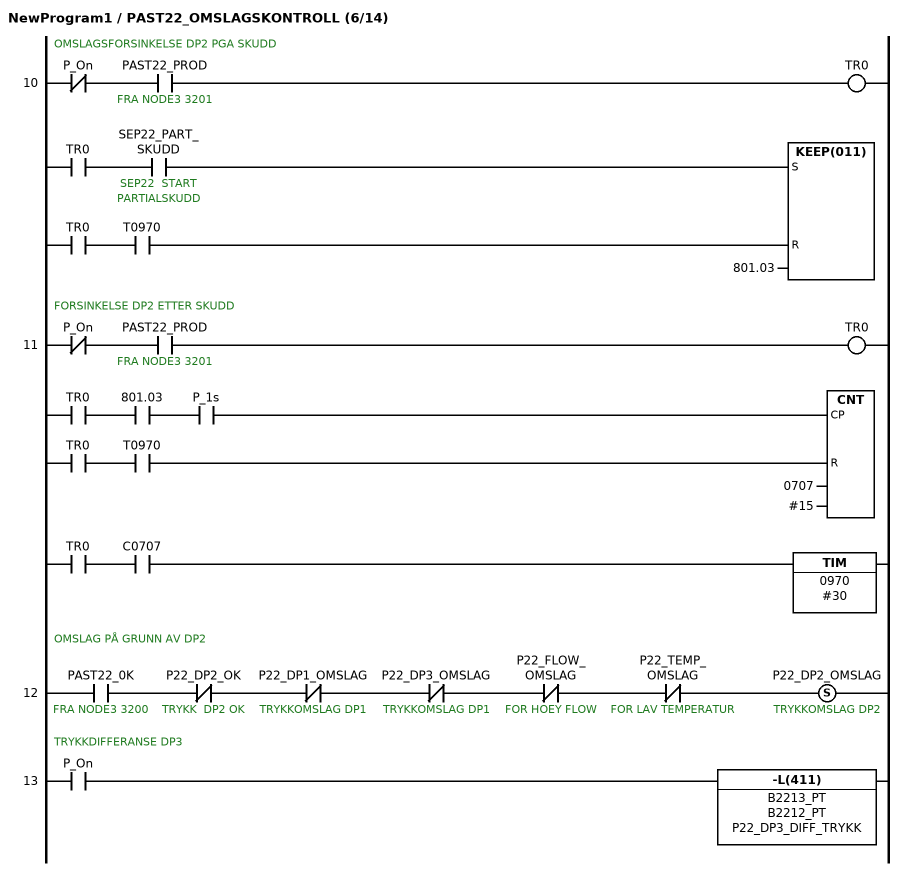
; [picture p1152: NewProgram1 / PAST22_OMSLAGSKONTROLL, rungs 10-13]
; rung 10: OMSLAGSFORSINKELSE DP2 PGA SKUDD
LDNOT P_On
AND PAST22_PROD  ; FRA NODE3 3201
OUT TR0
AND SEP22_PART_SKUDD  ; SEP22  START PARTIALSKUDD
LD TR0
AND T0970
KEEP(011) 801.03
; rung 11: FORSINKELSE DP2 ETTER SKUDD
LDNOT P_On
AND PAST22_PROD  ; FRA NODE3 3201
OUT TR0
AND 801.03
AND P_1s
LD TR0
AND T0970
CNT 0707 #15
LD TR0
AND C0707
TIM 0970 #30
; rung 12: OMSLAG PÅ GRUNN AV DP2
LD PAST22_0K  ; FRA NODE3 3200
ANDNOT P22_DP2_OK  ; TRYKK  DP2 OK
ANDNOT P22_DP1_OMSLAG  ; TRYKKOMSLAG DP1
ANDNOT P22_DP3_OMSLAG  ; TRYKKOMSLAG DP1
ANDNOT P22_FLOW_OMSLAG  ; FOR HOEY FLOW
ANDNOT P22_TEMP_OMSLAG  ; FOR LAV TEMPERATUR
SET P22_DP2_OMSLAG  ; TRYKKOMSLAG DP2
; rung 13: TRYKKDIFFERANSE DP3
LD P_On
-L(411) B2213_PT B2212_PT P22_DP3_DIFF_TRYKK

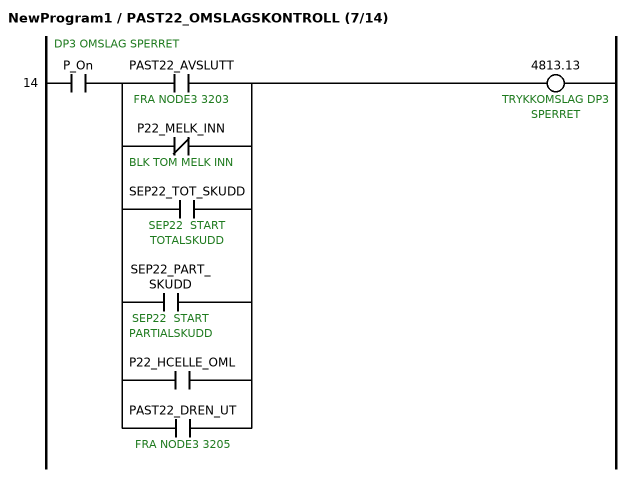
; rung 14: DP3 OMSLAG SPERRET
LD P_On  // CF113 INVERTERES OM SPERRING AV OMSLAG VED DP3 SKAL OPPHEVES
LD PAST22_AVSLUTT  ; FRA NODE3 3203
ORNOT P22_MELK_INN  ; BLK TOM MELK INN
OR SEP22_TOT_SKUDD  ; SEP22  START TOTALSKUDD
OR SEP22_PART_SKUDD  ; SEP22  START PARTIALSKUDD
OR P22_HCELLE_OML
OR PAST22_DREN_UT  ; FRA NODE3 3205
ANDLD
OUT 4813.13  ; TRYKKOMSLAG DP3 SPERRET

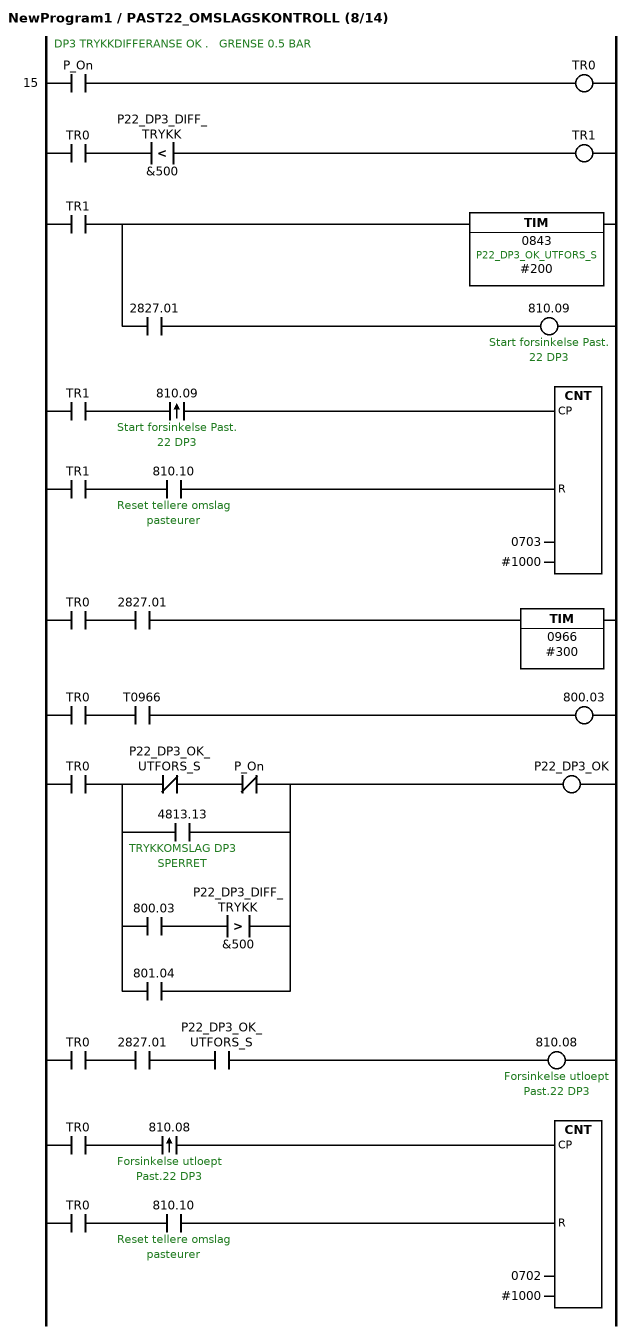
; rung 15: DP3 TRYKKDIFFERANSE OK .   GRENSE 0.5 BAR
LD P_On
OUT TR0
AND<SL(313) P22_DP3_DIFF_TRYKK &500
OUT TR1
TIM 0843 #200  ; P22_DP3_OK_UTFORS_S
AND 2827.01
OUT 810.09  ; Start forsinkelse Past. 22 DP3
LD TR1
@AND 810.09  ; Start forsinkelse Past. 22 DP3
LD TR1
AND 810.10  ; Reset tellere omslag pasteurer
CNT 0703 #1000
LD TR0
AND 2827.01
TIM 0966 #300
LD TR0
AND T0966
OUT 800.03
LD TR0
LDNOT P22_DP3_OK_UTFORS_S
ANDNOT P_On
OR 4813.13  ; TRYKKOMSLAG DP3 SPERRET
LD 800.03
AND>SL(323) P22_DP3_DIFF_TRYKK &500
ORLD
OR 801.04
ANDLD
OUT P22_DP3_OK
LD TR0
AND 2827.01
AND P22_DP3_OK_UTFORS_S
OUT 810.08  ; Forsinkelse utloept Past.22 DP3
LD TR0
@AND 810.08  ; Forsinkelse utloept Past.22 DP3
LD TR0
AND 810.10  ; Reset tellere omslag pasteurer
CNT 0702 #1000

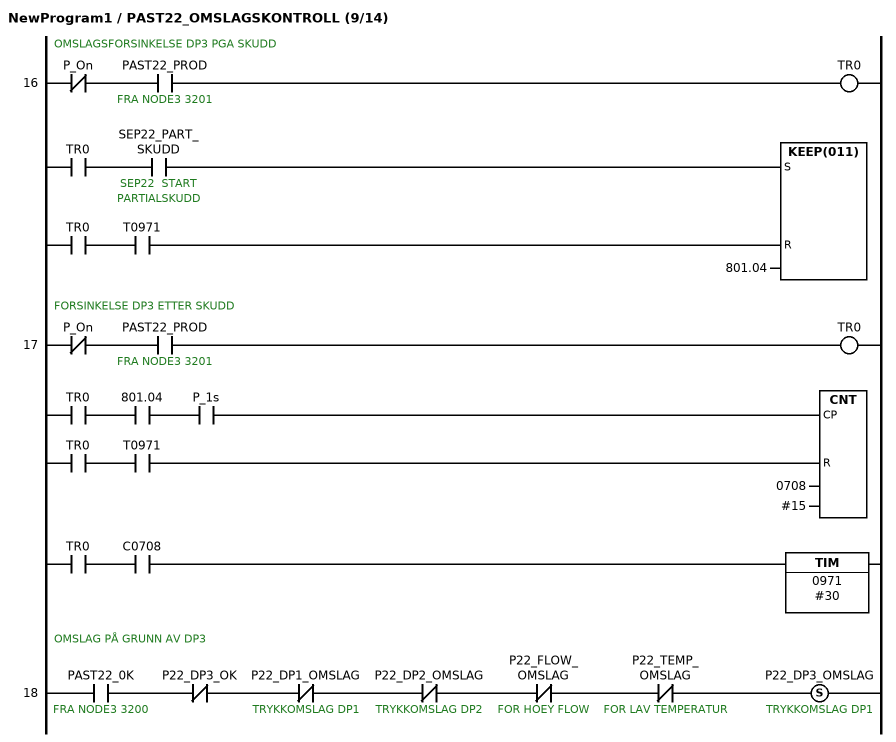
; rung 16: OMSLAGSFORSINKELSE DP3 PGA SKUDD
LDNOT P_On
AND PAST22_PROD  ; FRA NODE3 3201
OUT TR0
AND SEP22_PART_SKUDD  ; SEP22  START PARTIALSKUDD
LD TR0
AND T0971
KEEP(011) 801.04
; rung 17: FORSINKELSE DP3 ETTER SKUDD
LDNOT P_On
AND PAST22_PROD  ; FRA NODE3 3201
OUT TR0
AND 801.04
AND P_1s
LD TR0
AND T0971
CNT 0708 #15
LD TR0
AND C0708
TIM 0971 #30
; rung 18: OMSLAG PÅ GRUNN AV DP3
LD PAST22_0K  ; FRA NODE3 3200
ANDNOT P22_DP3_OK
ANDNOT P22_DP1_OMSLAG  ; TRYKKOMSLAG DP1
ANDNOT P22_DP2_OMSLAG  ; TRYKKOMSLAG DP2
ANDNOT P22_FLOW_OMSLAG  ; FOR HOEY FLOW
ANDNOT P22_TEMP_OMSLAG  ; FOR LAV TEMPERATUR
SET P22_DP3_OMSLAG  ; TRYKKOMSLAG DP1

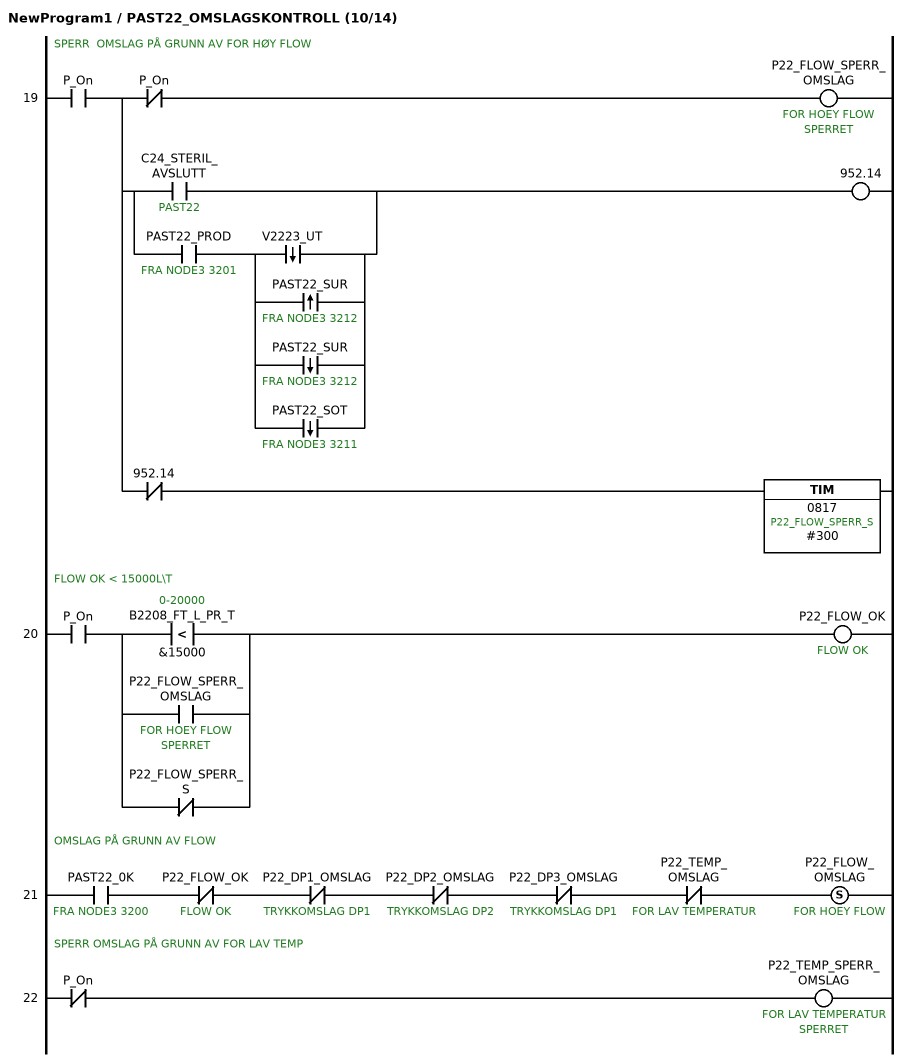
; rung 19: SPERR  OMSLAG PÅ GRUNN AV FOR HØY FLOW
LD P_On
OUT TR0
ANDNOT P_On  // CF113 INVERTERES OM SPERRING AV OMSLAG VED FOR HØY FLOW SKAL OPPHEVES
OUT P22_FLOW_SPERR_OMSLAG  ; FOR HOEY FLOW SPERRET
LD TR0
LD C24_STERIL_AVSLUTT  ; PAST22
LD PAST22_PROD  ; FRA NODE3 3201
%LD V2223_UT
@OR PAST22_SUR  ; FRA NODE3 3212
%OR PAST22_SUR  ; FRA NODE3 3212
%OR PAST22_SOT  ; FRA NODE3 3211
ANDLD
ORLD
ANDLD
OUT 952.14
LD TR0
ANDNOT 952.14
TIM 0817 #300  ; P22_FLOW_SPERR_S
; rung 20: FLOW OK < 15000L\T
LD P_On
LD<(310) B2208_FT_L_PR_T &15000  ; 0-20000
OR P22_FLOW_SPERR_OMSLAG  ; FOR HOEY FLOW SPERRET
ORNOT P22_FLOW_SPERR_S
ANDLD
OUT P22_FLOW_OK  ; FLOW OK
; rung 21: OMSLAG PÅ GRUNN AV FLOW
LD PAST22_0K  ; FRA NODE3 3200
ANDNOT P22_FLOW_OK  ; FLOW OK
ANDNOT P22_DP1_OMSLAG  ; TRYKKOMSLAG DP1
ANDNOT P22_DP2_OMSLAG  ; TRYKKOMSLAG DP2
ANDNOT P22_DP3_OMSLAG  ; TRYKKOMSLAG DP1
ANDNOT P22_TEMP_OMSLAG  ; FOR LAV TEMPERATUR
SET P22_FLOW_OMSLAG  ; FOR HOEY FLOW
; rung 22: SPERR OMSLAG PÅ GRUNN AV FOR LAV TEMP
LDNOT P_On  // CF113 INVERTERES OM SPERRING AV OMSLAG VED FOR LAV OMSLAGSTEMPERATUR
OUT P22_TEMP_SPERR_OMSLAG  ; FOR LAV TEMPERATUR SPERRET

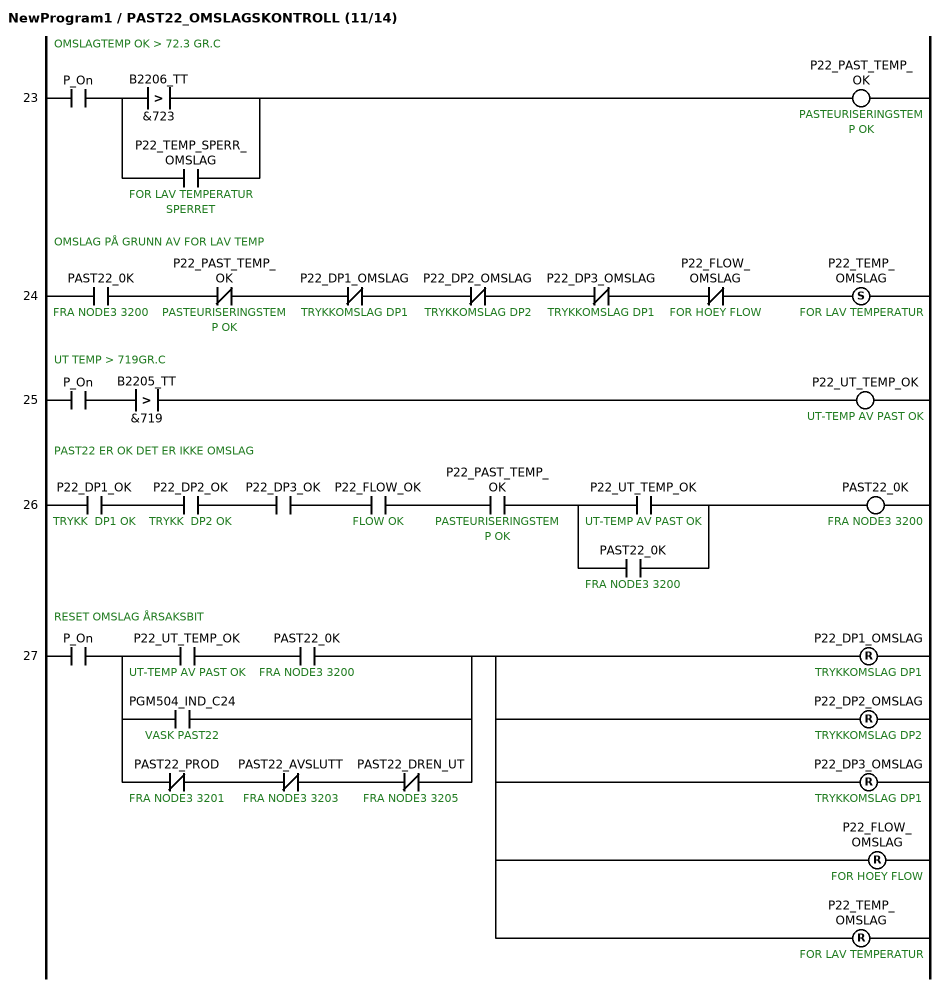
; rung 23: OMSLAGTEMP OK > 72.3 GR.C
LD P_On
LD>(320) B2206_TT &723
OR P22_TEMP_SPERR_OMSLAG  ; FOR LAV TEMPERATUR SPERRET
ANDLD
OUT P22_PAST_TEMP_OK  ; PASTEURISERINGSTEMP OK
; rung 24: OMSLAG PÅ GRUNN AV FOR LAV TEMP
LD PAST22_0K  ; FRA NODE3 3200
ANDNOT P22_PAST_TEMP_OK  ; PASTEURISERINGSTEMP OK
ANDNOT P22_DP1_OMSLAG  ; TRYKKOMSLAG DP1
ANDNOT P22_DP2_OMSLAG  ; TRYKKOMSLAG DP2
ANDNOT P22_DP3_OMSLAG  ; TRYKKOMSLAG DP1
ANDNOT P22_FLOW_OMSLAG  ; FOR HOEY FLOW
SET P22_TEMP_OMSLAG  ; FOR LAV TEMPERATUR
; rung 25: UT TEMP > 719GR.C
LD P_On
AND>(320) B2205_TT &719
OUT P22_UT_TEMP_OK  ; UT-TEMP AV PAST OK
; rung 26: PAST22 ER OK DET ER IKKE OMSLAG
LD P22_DP1_OK  ; TRYKK  DP1 OK
AND P22_DP2_OK  ; TRYKK  DP2 OK
AND P22_DP3_OK
AND P22_FLOW_OK  ; FLOW OK
AND P22_PAST_TEMP_OK  ; PASTEURISERINGSTEMP OK
LD P22_UT_TEMP_OK  ; UT-TEMP AV PAST OK
OR PAST22_0K  ; FRA NODE3 3200
ANDLD
OUT PAST22_0K  ; FRA NODE3 3200
; rung 27: RESET OMSLAG ÅRSAKSBIT
LD P_On
LD P22_UT_TEMP_OK  ; UT-TEMP AV PAST OK
AND PAST22_0K  ; FRA NODE3 3200
OR PGM504_IND_C24  ; VASK PAST22
LDNOT PAST22_PROD  ; FRA NODE3 3201
ANDNOT PAST22_AVSLUTT  ; FRA NODE3 3203
ANDNOT PAST22_DREN_UT  ; FRA NODE3 3205
ORLD
ANDLD
RSET P22_DP1_OMSLAG  ; TRYKKOMSLAG DP1
RSET P22_DP2_OMSLAG  ; TRYKKOMSLAG DP2
RSET P22_DP3_OMSLAG  ; TRYKKOMSLAG DP1
RSET P22_FLOW_OMSLAG  ; FOR HOEY FLOW
RSET P22_TEMP_OMSLAG  ; FOR LAV TEMPERATUR

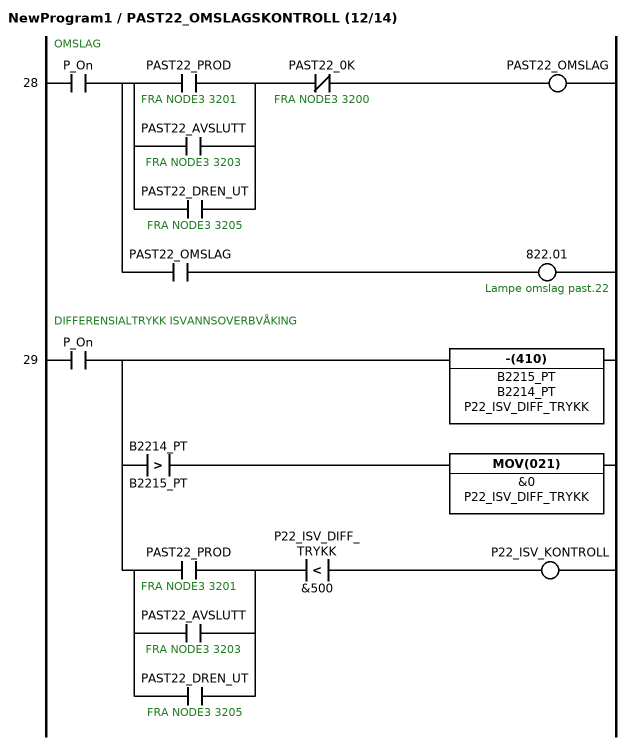
; rung 28: OMSLAG
LD P_On
OUT TR0
LD PAST22_PROD  ; FRA NODE3 3201
OR PAST22_AVSLUTT  ; FRA NODE3 3203
OR PAST22_DREN_UT  ; FRA NODE3 3205
ANDLD
ANDNOT PAST22_0K  ; FRA NODE3 3200
OUT PAST22_OMSLAG
LD TR0
AND PAST22_OMSLAG
OUT 822.01  ; Lampe omslag past.22
; rung 29: DIFFERENSIALTRYKK ISVANNSOVERBVÅKING
LD P_On
OUT TR0
-(410) B2215_PT B2214_PT P22_ISV_DIFF_TRYKK
AND>(320) B2214_PT B2215_PT
MOV(021) &0 P22_ISV_DIFF_TRYKK
LD TR0
LD PAST22_PROD  ; FRA NODE3 3201
OR PAST22_AVSLUTT  ; FRA NODE3 3203
OR PAST22_DREN_UT  ; FRA NODE3 3205
ANDLD
AND<(310) P22_ISV_DIFF_TRYKK &500
OUT P22_ISV_KONTROLL

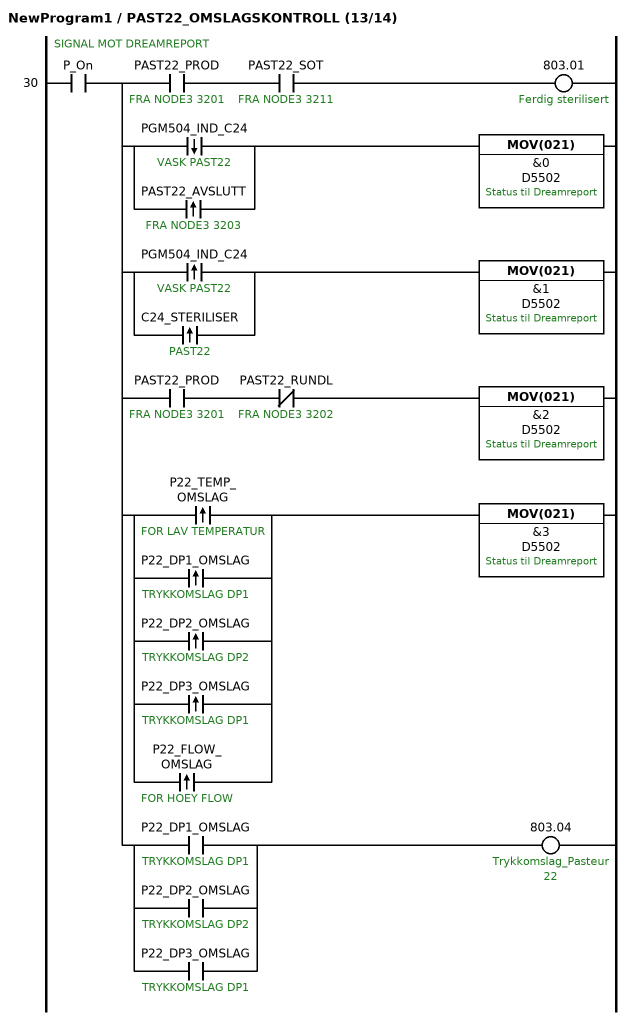
; rung 30: SIGNAL MOT DREAMREPORT
LD P_On
OUT TR0
AND PAST22_PROD  ; FRA NODE3 3201
AND PAST22_SOT  ; FRA NODE3 3211
OUT 803.01  ; Ferdig sterilisert
LD TR0
%LD PGM504_IND_C24  ; VASK PAST22
@OR PAST22_AVSLUTT  ; FRA NODE3 3203
ANDLD
MOV(021) &0 D5502  ; Status til Dreamreport
LD TR0
@LD PGM504_IND_C24  ; VASK PAST22
@OR C24_STERILISER  ; PAST22
ANDLD
MOV(021) &1 D5502  ; Status til Dreamreport
LD TR0
AND PAST22_PROD  ; FRA NODE3 3201
ANDNOT PAST22_RUNDL  ; FRA NODE3 3202
MOV(021) &2 D5502  ; Status til Dreamreport
LD TR0
@LD P22_TEMP_OMSLAG  ; FOR LAV TEMPERATUR
@OR P22_DP1_OMSLAG  ; TRYKKOMSLAG DP1
@OR P22_DP2_OMSLAG  ; TRYKKOMSLAG DP2
@OR P22_DP3_OMSLAG  ; TRYKKOMSLAG DP1
@OR P22_FLOW_OMSLAG  ; FOR HOEY FLOW
ANDLD
MOV(021) &3 D5502  ; Status til Dreamreport
LD TR0
LD P22_DP1_OMSLAG  ; TRYKKOMSLAG DP1
OR P22_DP2_OMSLAG  ; TRYKKOMSLAG DP2
OR P22_DP3_OMSLAG  ; TRYKKOMSLAG DP1
ANDLD
OUT 803.04  ; Trykkomslag_Pasteur 22

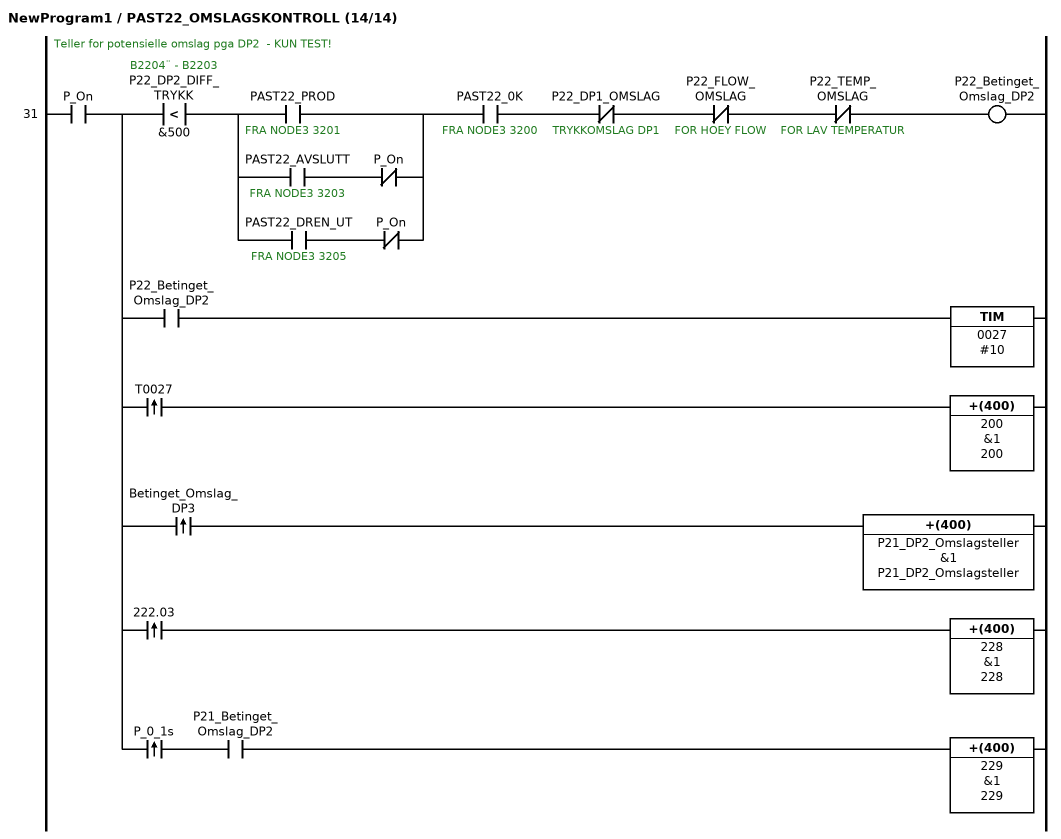
; rung 31: Teller for potensielle omslag pga DP2  - KUN TEST!
LD P_On
OUT TR0
AND<SL(313) P22_DP2_DIFF_TRYKK &500  ; B2204¨ - B2203
LD PAST22_PROD  ; FRA NODE3 3201
LD PAST22_AVSLUTT  ; FRA NODE3 3203
ANDNOT P_On
ORLD
LD PAST22_DREN_UT  ; FRA NODE3 3205
ANDNOT P_On
ORLD
ANDLD
AND PAST22_0K  ; FRA NODE3 3200
ANDNOT P22_DP1_OMSLAG  ; TRYKKOMSLAG DP1
ANDNOT P22_FLOW_OMSLAG  ; FOR HOEY FLOW
ANDNOT P22_TEMP_OMSLAG  ; FOR LAV TEMPERATUR
OUT P22_Betinget_Omslag_DP2
LD TR0
AND P22_Betinget_Omslag_DP2
TIM 0027 #10
LD TR0
@AND T0027
+(400) 200 &1 200
LD TR0
@AND Betinget_Omslag_DP3
+(400) P21_DP2_Omslagsteller &1 P21_DP2_Omslagsteller
LD TR0
@AND 222.03
+(400) 228 &1 228
LD TR0
@AND P_0_1s
AND P21_Betinget_Omslag_DP2
+(400) 229 &1 229

### Section PAST_22_TELLERFUNKSJONER

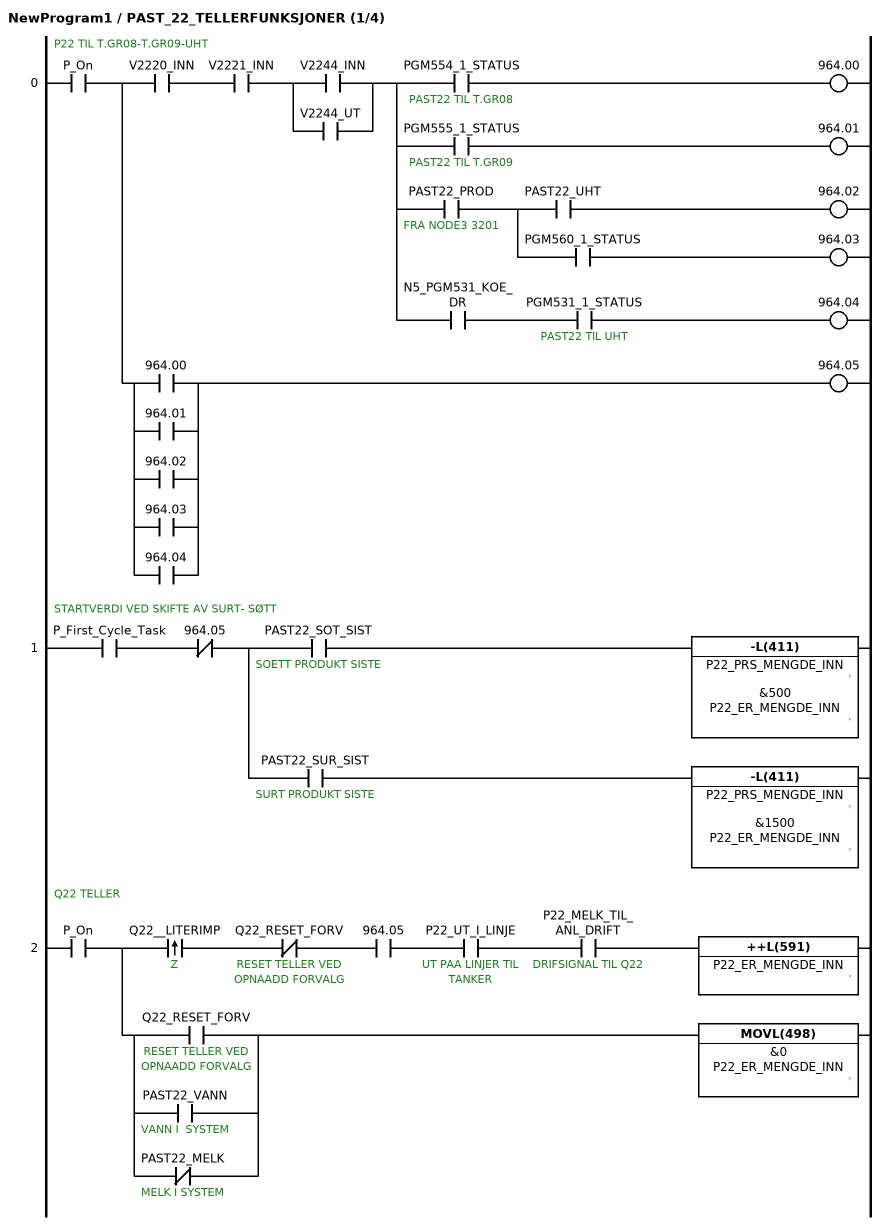
; rung 0: P22 TIL T.GR08-T.GR09-UHT
LD P_On
OUT TR0
AND V2220_INN
AND V2221_INN
LD V2244_INN
OR V2244_UT
ANDLD
OUT TR1
AND PGM554_1_STATUS  ; PAST22 TIL T.GR08
OUT 964.00
LD TR1
AND PGM555_1_STATUS  ; PAST22 TIL T.GR09
OUT 964.01
LD TR1
AND PAST22_PROD  ; FRA NODE3 3201
OUT TR2
AND PAST22_UHT
OUT 964.02
LD TR2
AND PGM560_1_STATUS
OUT 964.03
LD TR1
AND N5_PGM531_KOE_DR
AND PGM531_1_STATUS  ; PAST22 TIL UHT
OUT 964.04
LD TR0
LD 964.00
OR 964.01
OR 964.02
OR 964.03
OR 964.04
ANDLD
OUT 964.05
; rung 1: STARTVERDI VED SKIFTE AV SURT- SØTT
LD P_First_Cycle_Task
ANDNOT 964.05
OUT TR0
AND PAST22_SOT_SIST  ; SOETT PRODUKT SISTE
-L(411) P22_PRS_MENGDE_INN &500 P22_ER_MENGDE_INN  ; '
LD TR0
AND PAST22_SUR_SIST  ; SURT PRODUKT SISTE
-L(411) P22_PRS_MENGDE_INN &1500 P22_ER_MENGDE_INN  ; '
; rung 2: Q22 TELLER
LD P_On
OUT TR0
@AND Q22__LITERIMP  ; Z
ANDNOT Q22_RESET_FORV  ; RESET TELLER VED OPNAADD FORVALG
AND 964.05
AND P22_UT_I_LINJE  ; UT PAA LINJER TIL TANKER
AND P22_MELK_TIL_ANL_DRIFT  ; DRIFSIGNAL TIL Q22
++L(591) P22_ER_MENGDE_INN  ; '
LD TR0
LD Q22_RESET_FORV  ; RESET TELLER VED OPNAADD FORVALG
OR PAST22_VANN  ; VANN I  SYSTEM
ORNOT PAST22_MELK  ; MELK I SYSTEM
ANDLD
MOVL(498) &0 P22_ER_MENGDE_INN  ; '

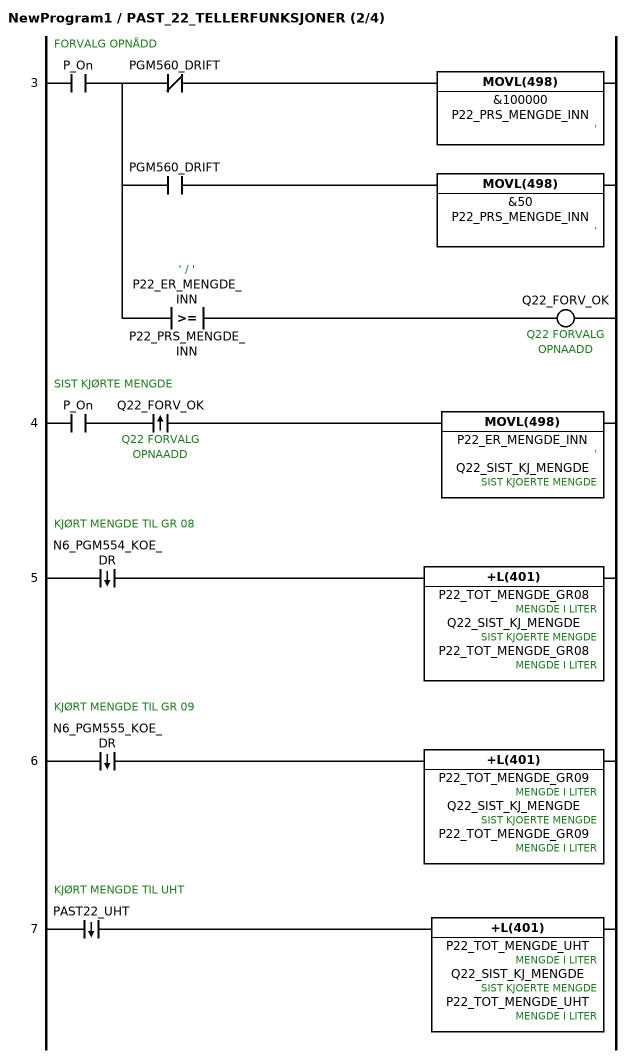
; rung 3: FORVALG OPNÅDD
LD P_On
OUT TR0
ANDNOT PGM560_DRIFT
MOVL(498) &100000 P22_PRS_MENGDE_INN  ; '
LD TR0
AND PGM560_DRIFT
MOVL(498) &50 P22_PRS_MENGDE_INN  ; '
LD TR0
AND>=L(326) P22_ER_MENGDE_INN P22_PRS_MENGDE_INN  ; '
OUT Q22_FORV_OK  ; Q22 FORVALG OPNAADD
; rung 4: SIST KJØRTE MENGDE
LD P_On
@AND Q22_FORV_OK  ; Q22 FORVALG OPNAADD
MOVL(498) P22_ER_MENGDE_INN Q22_SIST_KJ_MENGDE  ; ', SIST KJOERTE MENGDE
; rung 5: KJØRT MENGDE TIL GR 08
%LD N6_PGM554_KOE_DR
+L(401) P22_TOT_MENGDE_GR08 Q22_SIST_KJ_MENGDE P22_TOT_MENGDE_GR08  ; MENGDE I LITER, SIST KJOERTE MENGDE
; rung 6: KJØRT MENGDE TIL GR 09
%LD N6_PGM555_KOE_DR
+L(401) P22_TOT_MENGDE_GR09 Q22_SIST_KJ_MENGDE P22_TOT_MENGDE_GR09  ; MENGDE I LITER, SIST KJOERTE MENGDE
; rung 7: KJØRT MENGDE TIL UHT
%LD PAST22_UHT
+L(401) P22_TOT_MENGDE_UHT Q22_SIST_KJ_MENGDE P22_TOT_MENGDE_UHT  ; MENGDE I LITER, SIST KJOERTE MENGDE

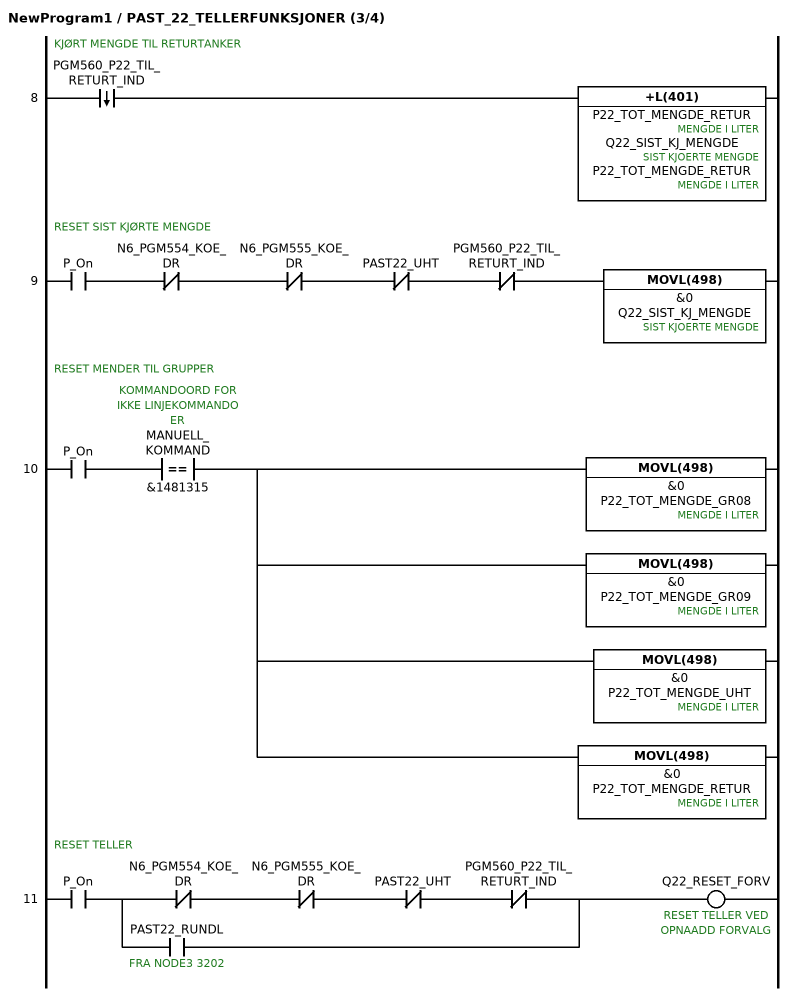
; rung 8: KJØRT MENGDE TIL RETURTANKER
%LD PGM560_P22_TIL_RETURT_IND
+L(401) P22_TOT_MENGDE_RETUR Q22_SIST_KJ_MENGDE P22_TOT_MENGDE_RETUR  ; MENGDE I LITER, SIST KJOERTE MENGDE
; rung 9: RESET SIST KJØRTE MENGDE
LD P_On
ANDNOT N6_PGM554_KOE_DR
ANDNOT N6_PGM555_KOE_DR
ANDNOT PAST22_UHT
ANDNOT PGM560_P22_TIL_RETURT_IND
MOVL(498) &0 Q22_SIST_KJ_MENGDE  ; SIST KJOERTE MENGDE
; rung 10: RESET MENDER TIL GRUPPER
LD P_On
AND=L(301) MANUELL_KOMMAND &1481315  ; KOMMANDOORD FOR IKKE LINJEKOMMANDOER
MOVL(498) &0 P22_TOT_MENGDE_GR08  ; MENGDE I LITER
MOVL(498) &0 P22_TOT_MENGDE_GR09  ; MENGDE I LITER
MOVL(498) &0 P22_TOT_MENGDE_UHT  ; MENGDE I LITER
MOVL(498) &0 P22_TOT_MENGDE_RETUR  ; MENGDE I LITER
; rung 11: RESET TELLER
LD P_On
LDNOT N6_PGM554_KOE_DR
ANDNOT N6_PGM555_KOE_DR
ANDNOT PAST22_UHT
ANDNOT PGM560_P22_TIL_RETURT_IND
OR PAST22_RUNDL  ; FRA NODE3 3202
ANDLD
OUT Q22_RESET_FORV  ; RESET TELLER VED OPNAADD FORVALG

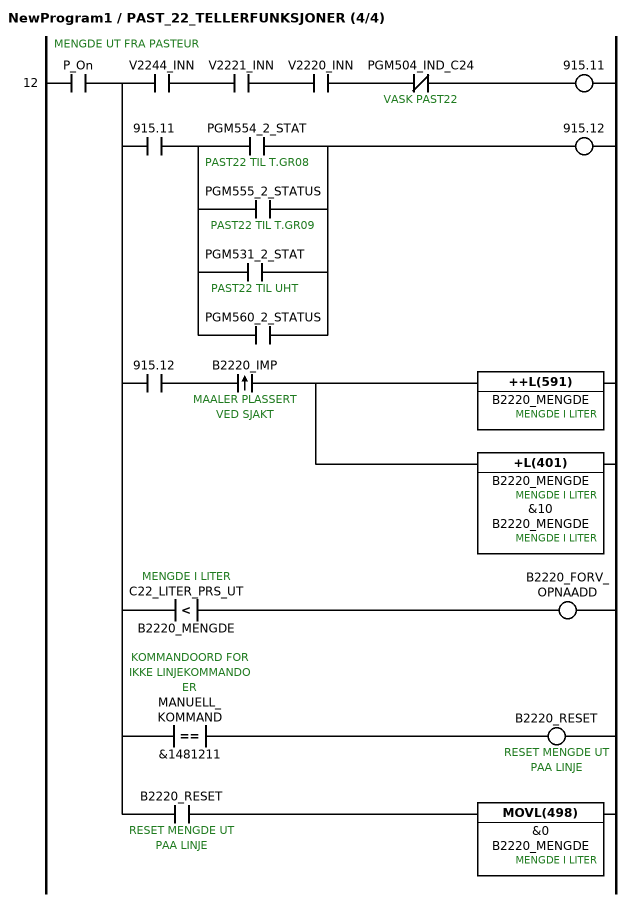
; rung 12: MENGDE UT FRA PASTEUR
LD P_On
OUT TR0
AND V2244_INN
AND V2221_INN
AND V2220_INN
ANDNOT PGM504_IND_C24  ; VASK PAST22
OUT 915.11
LD TR0
AND 915.11
LD PGM554_2_STAT  ; PAST22 TIL T.GR08
OR PGM555_2_STATUS  ; PAST22 TIL T.GR09
OR PGM531_2_STAT  ; PAST22 TIL UHT
OR PGM560_2_STATUS
ANDLD
OUT 915.12
LD TR0
AND 915.12
@AND B2220_IMP  ; MAALER PLASSERT VED SJAKT
++L(591) B2220_MENGDE  ; MENGDE I LITER
+L(401) B2220_MENGDE &10 B2220_MENGDE  ; MENGDE I LITER
LD TR0
AND<L(311) C22_LITER_PRS_UT B2220_MENGDE  ; MENGDE I LITER
OUT B2220_FORV_OPNAADD
LD TR0
AND=L(301) MANUELL_KOMMAND &1481211  ; KOMMANDOORD FOR IKKE LINJEKOMMANDOER
OUT B2220_RESET  ; RESET MENGDE UT PAA LINJE
LD TR0
AND B2220_RESET  ; RESET MENGDE UT PAA LINJE
MOVL(498) &0 B2220_MENGDE  ; MENGDE I LITER

### Section P22_MELK_IRØR_TIL_TGR

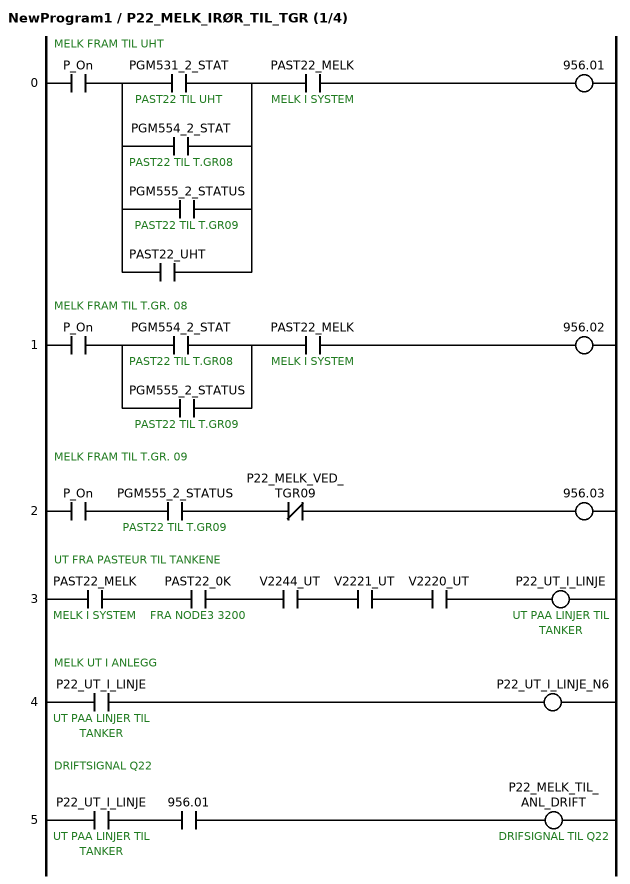
; rung 0: MELK FRAM TIL UHT
LD P_On
LD PGM531_2_STAT  ; PAST22 TIL UHT
OR PGM554_2_STAT  ; PAST22 TIL T.GR08
OR PGM555_2_STATUS  ; PAST22 TIL T.GR09
OR PAST22_UHT
ANDLD
AND PAST22_MELK  ; MELK I SYSTEM
OUT 956.01
; rung 1: MELK FRAM TIL T.GR. 08
LD P_On
LD PGM554_2_STAT  ; PAST22 TIL T.GR08
OR PGM555_2_STATUS  ; PAST22 TIL T.GR09
ANDLD
AND PAST22_MELK  ; MELK I SYSTEM
OUT 956.02
; rung 2: MELK FRAM TIL T.GR. 09
LD P_On
AND PGM555_2_STATUS  ; PAST22 TIL T.GR09
ANDNOT P22_MELK_VED_TGR09
OUT 956.03
; rung 3: UT FRA PASTEUR TIL TANKENE
LD PAST22_MELK  ; MELK I SYSTEM
AND PAST22_0K  ; FRA NODE3 3200
AND V2244_UT
AND V2221_UT
AND V2220_UT
OUT P22_UT_I_LINJE  ; UT PAA LINJER TIL TANKER
; rung 4: MELK UT I ANLEGG
LD P22_UT_I_LINJE  ; UT PAA LINJER TIL TANKER
OUT P22_UT_I_LINJE_N6
; rung 5: DRIFTSIGNAL Q22
LD P22_UT_I_LINJE  ; UT PAA LINJER TIL TANKER
AND 956.01
OUT P22_MELK_TIL_ANL_DRIFT  ; DRIFSIGNAL TIL Q22

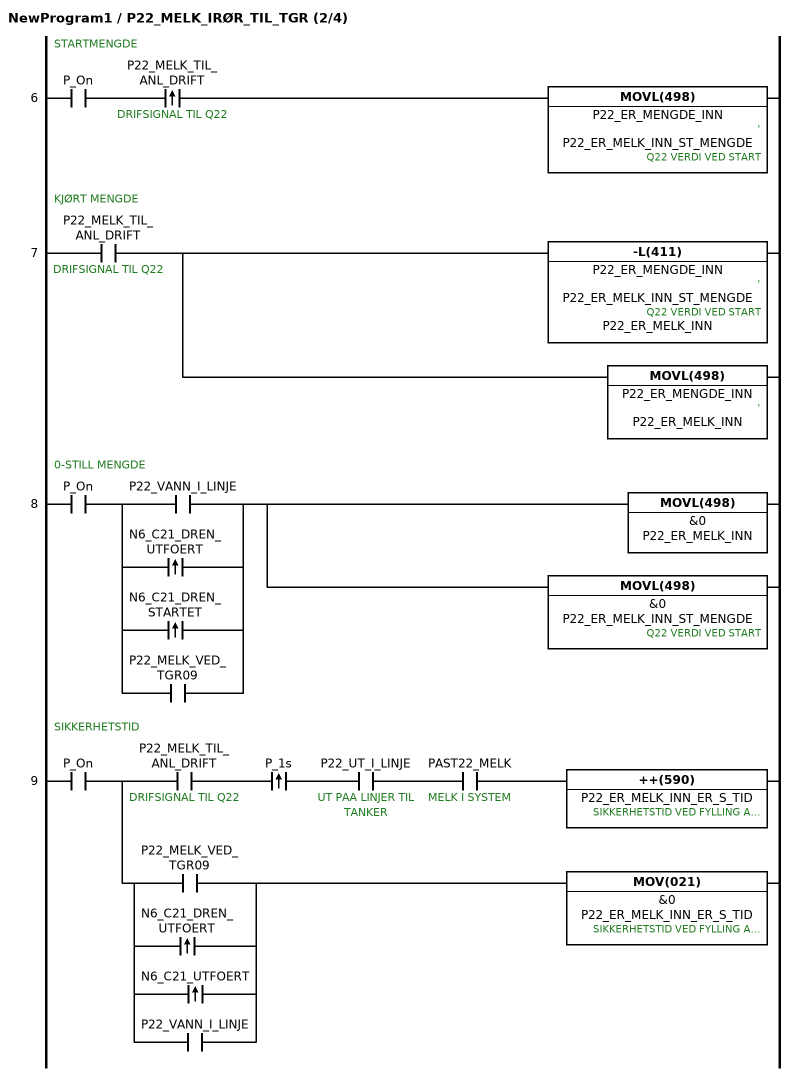
; rung 6: STARTMENGDE
LD P_On
@AND P22_MELK_TIL_ANL_DRIFT  ; DRIFSIGNAL TIL Q22
MOVL(498) P22_ER_MENGDE_INN P22_ER_MELK_INN_ST_MENGDE  ; ', Q22 VERDI VED START
; rung 7: KJØRT MENGDE
LD P22_MELK_TIL_ANL_DRIFT  ; DRIFSIGNAL TIL Q22
-L(411) P22_ER_MENGDE_INN P22_ER_MELK_INN_ST_MENGDE P22_ER_MELK_INN  ; ', Q22 VERDI VED START
MOVL(498) P22_ER_MENGDE_INN P22_ER_MELK_INN  ; '
; rung 8: 0-STILL MENGDE
LD P_On
LD P22_VANN_I_LINJE
@OR N6_C21_DREN_UTFOERT
@OR N6_C21_DREN_STARTET
OR P22_MELK_VED_TGR09
ANDLD
MOVL(498) &0 P22_ER_MELK_INN
MOVL(498) &0 P22_ER_MELK_INN_ST_MENGDE  ; Q22 VERDI VED START
; rung 9: SIKKERHETSTID
LD P_On
OUT TR0
AND P22_MELK_TIL_ANL_DRIFT  ; DRIFSIGNAL TIL Q22
@AND P_1s
AND P22_UT_I_LINJE  ; UT PAA LINJER TIL TANKER
AND PAST22_MELK  ; MELK I SYSTEM
++(590) P22_ER_MELK_INN_ER_S_TID  ; SIKKERHETSTID VED FYLLING AV MELK
LD TR0
LD P22_MELK_VED_TGR09
@OR N6_C21_DREN_UTFOERT
@OR N6_C21_UTFOERT
OR P22_VANN_I_LINJE
ANDLD
MOV(021) &0 P22_ER_MELK_INN_ER_S_TID  ; SIKKERHETSTID VED FYLLING AV MELK

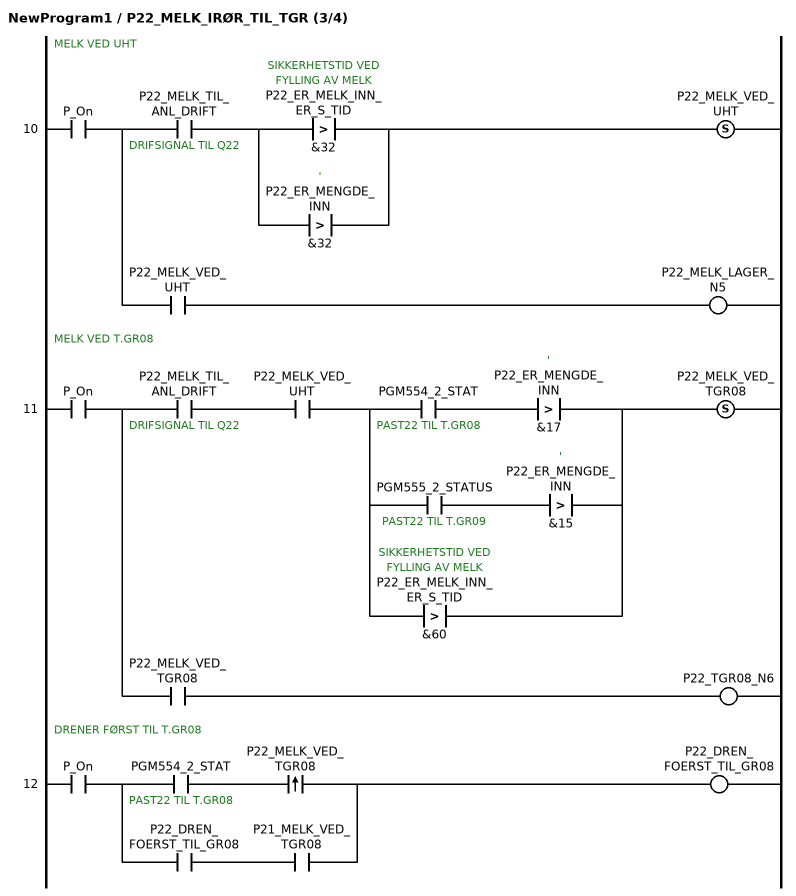
; rung 10: MELK VED UHT
LD P_On
OUT TR0
AND P22_MELK_TIL_ANL_DRIFT  ; DRIFSIGNAL TIL Q22
LD>(320) P22_ER_MELK_INN_ER_S_TID &32  ; SIKKERHETSTID VED FYLLING AV MELK
OR>(320) P22_ER_MENGDE_INN &32  ; '
ANDLD
SET P22_MELK_VED_UHT
LD TR0
AND P22_MELK_VED_UHT
OUT P22_MELK_LAGER_N5
; rung 11: MELK VED T.GR08
LD P_On
OUT TR0
AND P22_MELK_TIL_ANL_DRIFT  ; DRIFSIGNAL TIL Q22
AND P22_MELK_VED_UHT
LD PGM554_2_STAT  ; PAST22 TIL T.GR08
AND>L(321) P22_ER_MENGDE_INN &17  ; '
LD PGM555_2_STATUS  ; PAST22 TIL T.GR09
AND>L(321) P22_ER_MENGDE_INN &15  ; '
ORLD
OR>(320) P22_ER_MELK_INN_ER_S_TID &60  ; SIKKERHETSTID VED FYLLING AV MELK
ANDLD
SET P22_MELK_VED_TGR08
LD TR0
AND P22_MELK_VED_TGR08
OUT P22_TGR08_N6
; rung 12: DRENER FØRST TIL T.GR08
LD P_On
LD PGM554_2_STAT  ; PAST22 TIL T.GR08
@AND P22_MELK_VED_TGR08
LD P22_DREN_FOERST_TIL_GR08
AND P21_MELK_VED_TGR08
ORLD
ANDLD
OUT P22_DREN_FOERST_TIL_GR08

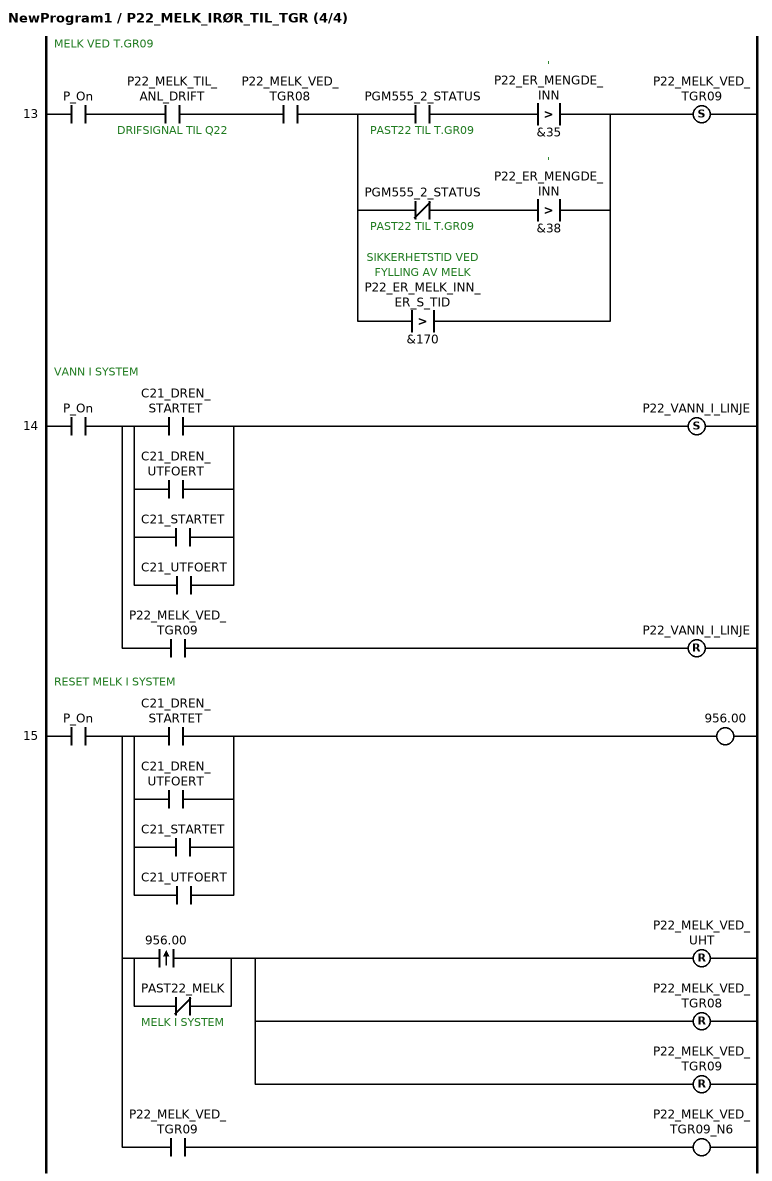
; rung 13: MELK VED T.GR09
LD P_On
AND P22_MELK_TIL_ANL_DRIFT  ; DRIFSIGNAL TIL Q22
AND P22_MELK_VED_TGR08
LD PGM555_2_STATUS  ; PAST22 TIL T.GR09
AND>L(321) P22_ER_MENGDE_INN &35  ; '
LDNOT PGM555_2_STATUS  ; PAST22 TIL T.GR09
AND>L(321) P22_ER_MENGDE_INN &38  ; '
ORLD
OR>(320) P22_ER_MELK_INN_ER_S_TID &170  ; SIKKERHETSTID VED FYLLING AV MELK
ANDLD
SET P22_MELK_VED_TGR09
; rung 14: VANN I SYSTEM
LD P_On
OUT TR0
LD C21_DREN_STARTET
OR C21_DREN_UTFOERT
OR C21_STARTET
OR C21_UTFOERT
ANDLD
SET P22_VANN_I_LINJE
LD TR0
AND P22_MELK_VED_TGR09
RSET P22_VANN_I_LINJE
; rung 15: RESET MELK I SYSTEM
LD P_On
OUT TR0
LD C21_DREN_STARTET
OR C21_DREN_UTFOERT
OR C21_STARTET
OR C21_UTFOERT
ANDLD
OUT 956.00
LD TR0
@LD 956.00
ORNOT PAST22_MELK  ; MELK I SYSTEM
ANDLD
RSET P22_MELK_VED_UHT
RSET P22_MELK_VED_TGR08
RSET P22_MELK_VED_TGR09
LD TR0
AND P22_MELK_VED_TGR09
OUT P22_MELK_VED_TGR09_N6

### Section P2201_FLOWKONTROLL

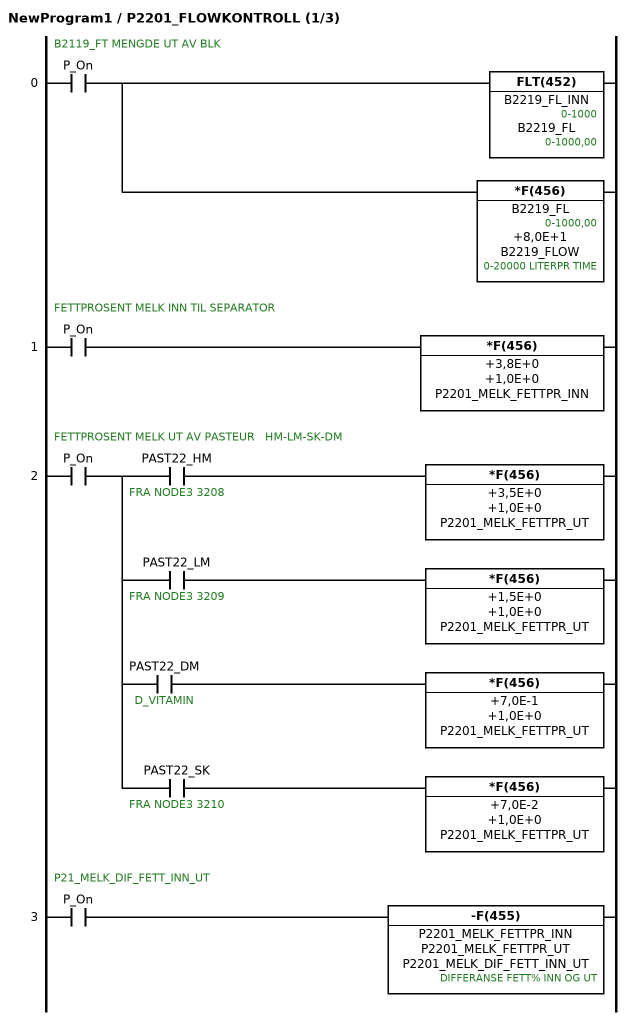
; rung 0: B2119_FT MENGDE UT AV BLK
LD P_On
FLT(452) B2219_FL_INN B2219_FL  ; 0-1000, 0-1000,00
*F(456) B2219_FL +8,0E+1 B2219_FLOW  ; 0-1000,00, 0-20000 LITERPR TIME
; rung 1: FETTPROSENT MELK INN TIL SEPARATOR
LD P_On
*F(456) +3,8E+0 +1,0E+0 P2201_MELK_FETTPR_INN
; rung 2: FETTPROSENT MELK UT AV PASTEUR   HM-LM-SK-DM
LD P_On
OUT TR0
AND PAST22_HM  ; FRA NODE3 3208
*F(456) +3,5E+0 +1,0E+0 P2201_MELK_FETTPR_UT
LD TR0
AND PAST22_LM  ; FRA NODE3 3209
*F(456) +1,5E+0 +1,0E+0 P2201_MELK_FETTPR_UT
LD TR0
AND PAST22_DM  ; D_VITAMIN
*F(456) +7,0E-1 +1,0E+0 P2201_MELK_FETTPR_UT
LD TR0
AND PAST22_SK  ; FRA NODE3 3210
*F(456) +7,0E-2 +1,0E+0 P2201_MELK_FETTPR_UT
; rung 3: P21_MELK_DIF_FETT_INN_UT
LD P_On
-F(455) P2201_MELK_FETTPR_INN P2201_MELK_FETTPR_UT P2201_MELK_DIF_FETT_INN_UT  ; DIFFERANSE FETT% INN OG UT

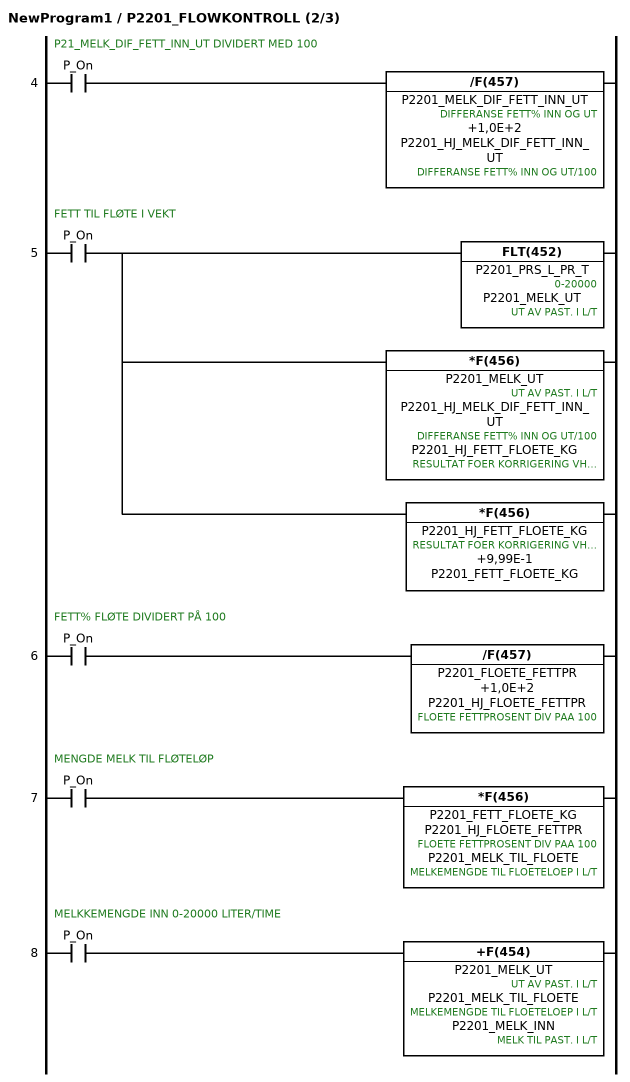
; rung 4: P21_MELK_DIF_FETT_INN_UT DIVIDERT MED 100
LD P_On
/F(457) P2201_MELK_DIF_FETT_INN_UT +1,0E+2 P2201_HJ_MELK_DIF_FETT_INN_UT  ; DIFFERANSE FETT% INN OG UT, DIFFERANSE FETT% INN OG UT/100
; rung 5: FETT TIL FLØTE I VEKT
LD P_On
FLT(452) P2201_PRS_L_PR_T P2201_MELK_UT  ; 0-20000, UT AV PAST. I L/T
*F(456) P2201_MELK_UT P2201_HJ_MELK_DIF_FETT_INN_UT P2201_HJ_FETT_FLOETE_KG  ; UT AV PAST. I L/T, DIFFERANSE FETT% INN OG UT/100, RESULTAT FOER KORRIGERING VHA EGENVEKT
*F(456) P2201_HJ_FETT_FLOETE_KG +9,99E-1 P2201_FETT_FLOETE_KG  ; RESULTAT FOER KORRIGERING VHA EGENVEKT
; rung 6: FETT% FLØTE DIVIDERT PÅ 100
LD P_On
/F(457) P2201_FLOETE_FETTPR +1,0E+2 P2201_HJ_FLOETE_FETTPR  ; FLOETE FETTPROSENT DIV PAA 100
; rung 7: MENGDE MELK TIL FLØTELØP
LD P_On
*F(456) P2201_FETT_FLOETE_KG P2201_HJ_FLOETE_FETTPR P2201_MELK_TIL_FLOETE  ; FLOETE FETTPROSENT DIV PAA 100, MELKEMENGDE TIL FLOETELOEP I L/T
; rung 8: MELKKEMENGDE INN 0-20000 LITER/TIME
LD P_On
+F(454) P2201_MELK_UT P2201_MELK_TIL_FLOETE P2201_MELK_INN  ; UT AV PAST. I L/T, MELKEMENGDE TIL FLOETELOEP I L/T, MELK TIL PAST. I L/T

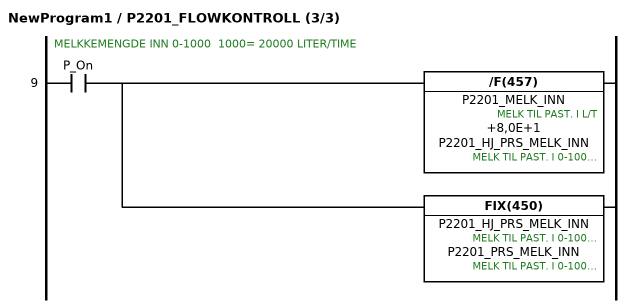
; rung 9: MELKKEMENGDE INN 0-1000  1000= 20000 LITER/TIME
LD P_On
/F(457) P2201_MELK_INN +8,0E+1 P2201_HJ_PRS_MELK_INN  ; MELK TIL PAST. I L/T, MELK TIL PAST. I 0-1000 1000=20000L/T
FIX(450) P2201_HJ_PRS_MELK_INN P2201_PRS_MELK_INN  ; MELK TIL PAST. I 0-1000 1000=20000L/T

### Section P2201

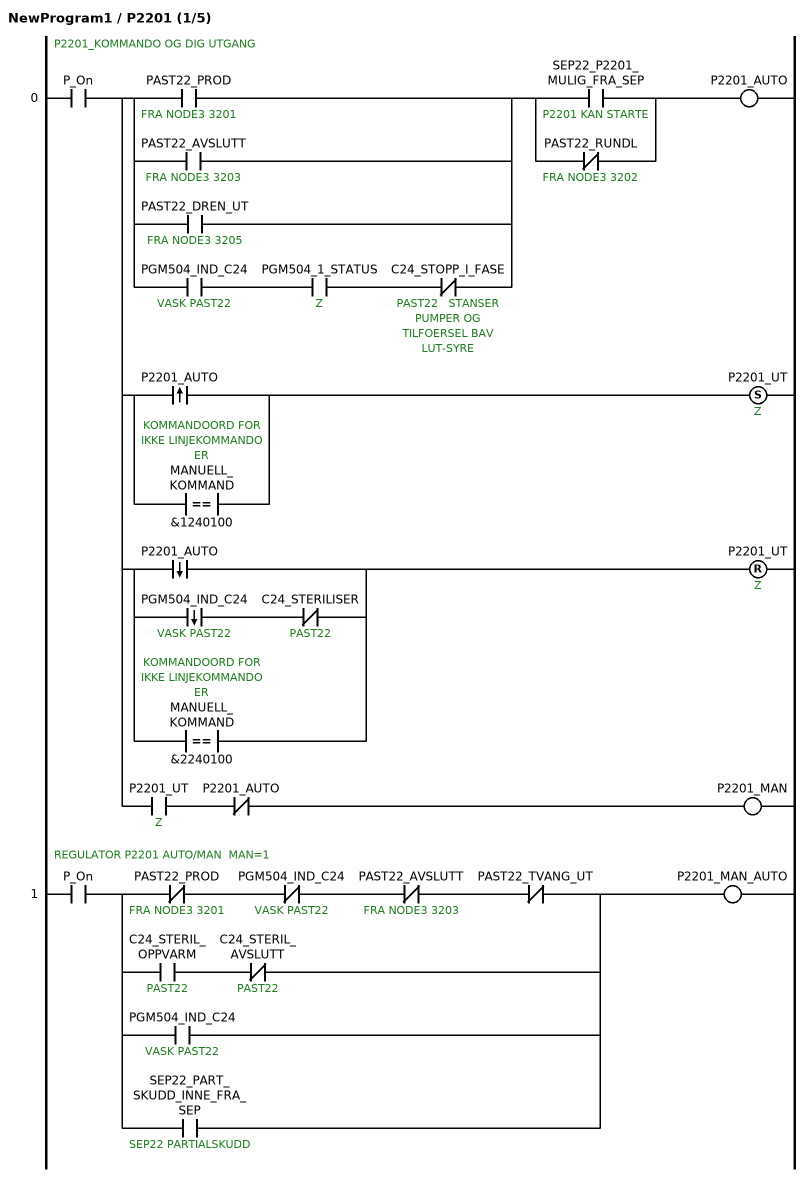
; rung 0: P2201_KOMMANDO OG DIG UTGANG
LD P_On
OUT TR0
LD PAST22_PROD  ; FRA NODE3 3201
OR PAST22_AVSLUTT  ; FRA NODE3 3203
OR PAST22_DREN_UT  ; FRA NODE3 3205
LD PGM504_IND_C24  ; VASK PAST22
AND PGM504_1_STATUS  ; Z
ANDNOT C24_STOPP_I_FASE  ; PAST22   STANSER PUMPER OG TILFOERSEL BAV LUT-SYRE
ORLD
ANDLD
LD SEP22_P2201_MULIG_FRA_SEP  ; P2201 KAN STARTE
ORNOT PAST22_RUNDL  ; FRA NODE3 3202
ANDLD
OUT P2201_AUTO
LD TR0
@LD P2201_AUTO
OR=L(301) MANUELL_KOMMAND &1240100  ; KOMMANDOORD FOR IKKE LINJEKOMMANDOER
ANDLD
SET P2201_UT  ; Z
LD TR0
%LD P2201_AUTO
%LD PGM504_IND_C24  ; VASK PAST22
ANDNOT C24_STERILISER  ; PAST22
ORLD
OR=L(301) MANUELL_KOMMAND &2240100  ; KOMMANDOORD FOR IKKE LINJEKOMMANDOER
ANDLD
RSET P2201_UT  ; Z
LD TR0
AND P2201_UT  ; Z
ANDNOT P2201_AUTO
OUT P2201_MAN
; rung 1: REGULATOR P2201 AUTO/MAN  MAN=1
LD P_On
LDNOT PAST22_PROD  ; FRA NODE3 3201
ANDNOT PGM504_IND_C24  ; VASK PAST22
ANDNOT PAST22_AVSLUTT  ; FRA NODE3 3203
ANDNOT PAST22_TVANG_UT
LD C24_STERIL_OPPVARM  ; PAST22
ANDNOT C24_STERIL_AVSLUTT  ; PAST22
ORLD
OR PGM504_IND_C24  ; VASK PAST22
OR SEP22_PART_SKUDD_INNE_FRA_SEP  ; SEP22 PARTIALSKUDD
ANDLD
OUT P2201_MAN_AUTO

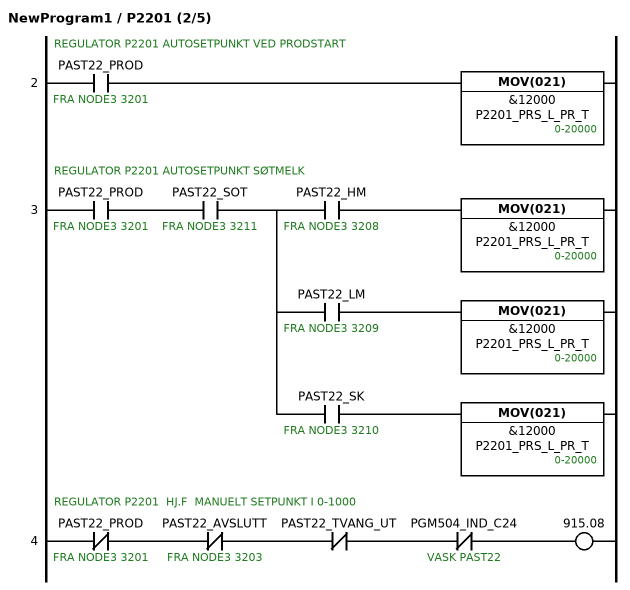
; rung 2: REGULATOR P2201 AUTOSETPUNKT VED PRODSTART
LD PAST22_PROD  ; FRA NODE3 3201
MOV(021) &12000 P2201_PRS_L_PR_T  ; 0-20000
; rung 3: REGULATOR P2201 AUTOSETPUNKT SØTMELK
LD PAST22_PROD  ; FRA NODE3 3201
AND PAST22_SOT  ; FRA NODE3 3211
OUT TR0
AND PAST22_HM  ; FRA NODE3 3208
MOV(021) &12000 P2201_PRS_L_PR_T  ; 0-20000
LD TR0
AND PAST22_LM  ; FRA NODE3 3209
MOV(021) &12000 P2201_PRS_L_PR_T  ; 0-20000
LD TR0
AND PAST22_SK  ; FRA NODE3 3210
MOV(021) &12000 P2201_PRS_L_PR_T  ; 0-20000
; rung 4: REGULATOR P2201  HJ.F  MANUELT SETPUNKT I 0-1000
LDNOT PAST22_PROD  ; FRA NODE3 3201
ANDNOT PAST22_AVSLUTT  ; FRA NODE3 3203
ANDNOT PAST22_TVANG_UT
ANDNOT PGM504_IND_C24  ; VASK PAST22
OUT 915.08

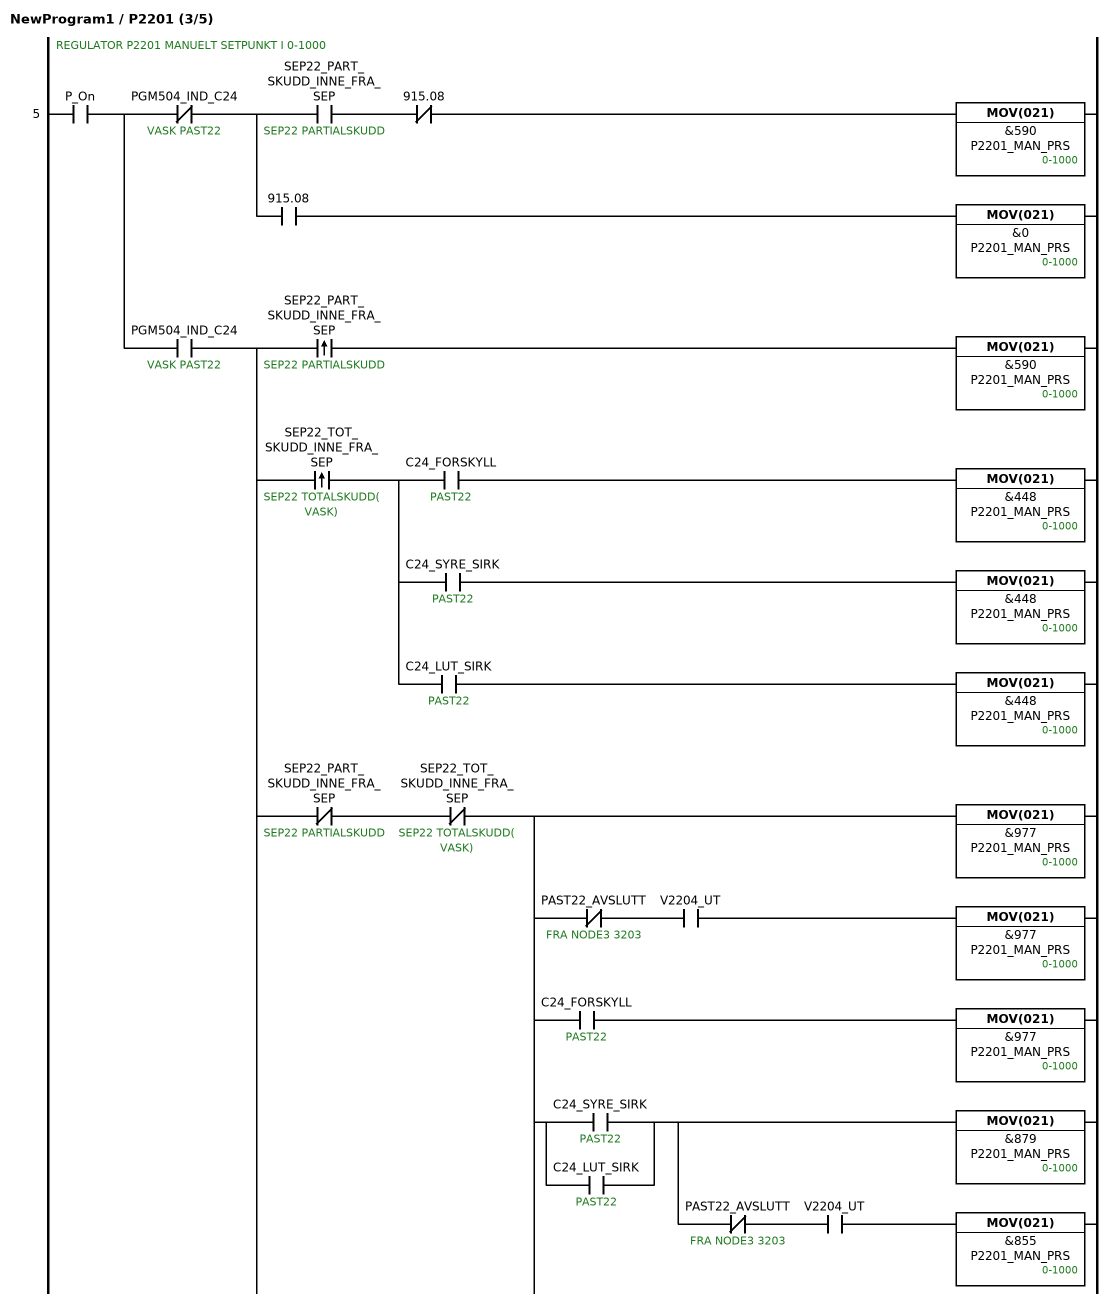

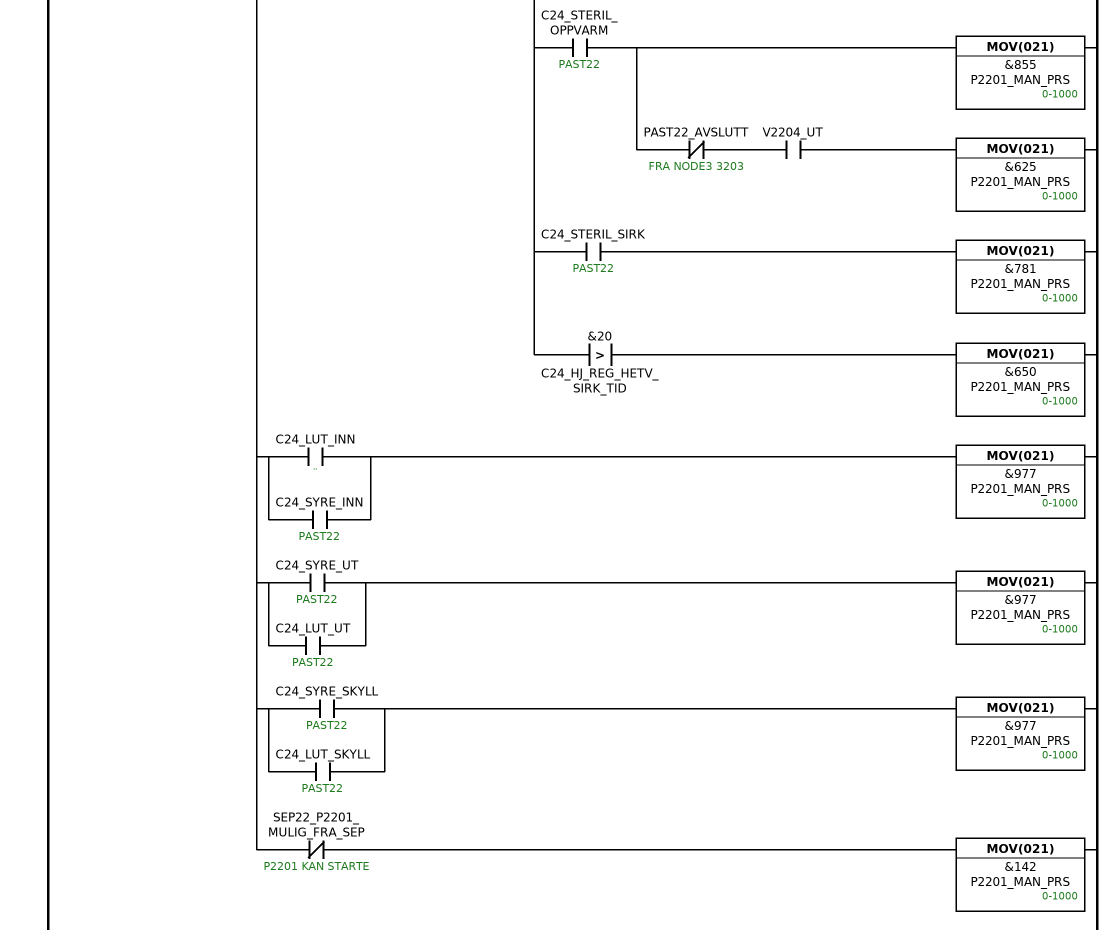
; rung 5: REGULATOR P2201 MANUELT SETPUNKT I 0-1000
LD P_On
OUT TR0
ANDNOT PGM504_IND_C24  ; VASK PAST22
OUT TR1
AND SEP22_PART_SKUDD_INNE_FRA_SEP  ; SEP22 PARTIALSKUDD
ANDNOT 915.08
MOV(021) &590 P2201_MAN_PRS  ; 0-1000
LD TR1
AND 915.08
MOV(021) &0 P2201_MAN_PRS  ; 0-1000
LD TR0
AND PGM504_IND_C24  ; VASK PAST22
OUT TR0
@AND SEP22_PART_SKUDD_INNE_FRA_SEP  ; SEP22 PARTIALSKUDD
MOV(021) &590 P2201_MAN_PRS  ; 0-1000
LD TR0
@AND SEP22_TOT_SKUDD_INNE_FRA_SEP  ; SEP22 TOTALSKUDD(VASK)
OUT TR1
AND C24_FORSKYLL  ; PAST22
MOV(021) &448 P2201_MAN_PRS  ; 0-1000
LD TR1
AND C24_SYRE_SIRK  ; PAST22
MOV(021) &448 P2201_MAN_PRS  ; 0-1000
LD TR1
AND C24_LUT_SIRK  ; PAST22
MOV(021) &448 P2201_MAN_PRS  ; 0-1000
LD TR0
ANDNOT SEP22_PART_SKUDD_INNE_FRA_SEP  ; SEP22 PARTIALSKUDD
ANDNOT SEP22_TOT_SKUDD_INNE_FRA_SEP  ; SEP22 TOTALSKUDD(VASK)
OUT TR1
MOV(021) &977 P2201_MAN_PRS  ; 0-1000
ANDNOT PAST22_AVSLUTT  ; FRA NODE3 3203
AND V2204_UT
MOV(021) &977 P2201_MAN_PRS  ; 0-1000
LD TR1
AND C24_FORSKYLL  ; PAST22
MOV(021) &977 P2201_MAN_PRS  ; 0-1000
LD TR1
LD C24_SYRE_SIRK  ; PAST22
OR C24_LUT_SIRK  ; PAST22
ANDLD
MOV(021) &879 P2201_MAN_PRS  ; 0-1000
ANDNOT PAST22_AVSLUTT  ; FRA NODE3 3203
AND V2204_UT
MOV(021) &855 P2201_MAN_PRS  ; 0-1000
LD TR1
AND C24_STERIL_OPPVARM  ; PAST22
MOV(021) &855 P2201_MAN_PRS  ; 0-1000
ANDNOT PAST22_AVSLUTT  ; FRA NODE3 3203
AND V2204_UT
MOV(021) &625 P2201_MAN_PRS  ; 0-1000
LD TR1
AND C24_STERIL_SIRK  ; PAST22
MOV(021) &781 P2201_MAN_PRS  ; 0-1000
LD TR1
AND>(320) &20 C24_HJ_REG_HETV_SIRK_TID
MOV(021) &650 P2201_MAN_PRS  ; 0-1000
LD TR0
LD C24_LUT_INN  ; ¨
OR C24_SYRE_INN  ; PAST22
ANDLD
MOV(021) &977 P2201_MAN_PRS  ; 0-1000
LD TR0
LD C24_SYRE_UT  ; PAST22
OR C24_LUT_UT  ; PAST22
ANDLD
MOV(021) &977 P2201_MAN_PRS  ; 0-1000
LD TR0
LD C24_SYRE_SKYLL  ; PAST22
OR C24_LUT_SKYLL  ; PAST22
ANDLD
MOV(021) &977 P2201_MAN_PRS  ; 0-1000
LD TR0
ANDNOT SEP22_P2201_MULIG_FRA_SEP  ; P2201 KAN STARTE
MOV(021) &142 P2201_MAN_PRS  ; 0-1000

